// TIA Portal V20 export
// export: Created 2026-04-28T10:05:06.6637609Z, ExportSetting WithDefaults, DisplayName Totally Integrated Automation Portal, DisplayVersion V20, DisplayName TIA Portal Openness, DisplayVersion V20, DisplayName TIA Portal Version Control Interface, DisplayVersion V20, DisplayName SINAMICS Startdrive Advanced, DisplayVersion V20, DisplayName SINAMICS Startdrive G130, G150, S120, S150, SINAMICS MV, G220, S200, S210, DisplayVersion V20, DisplayName SINAMICS Startdrive G110M, G120, G120C, G120D, G120P, G115D, DisplayVersion V20, DisplayName STEP 7 Professional, DisplayVersion V20, DisplayName STEP 7 Safety, DisplayVersion V20, DisplayName WinCC Basic/Comfort/Advanced, DisplayVersion V20, DisplayName WinCC Unified, DisplayVersion V20
TYPE "REZEPT_VisuDaten"
TITLE = Rezeptdaten-Visualisierung
// Dieser Datentyp beinhaltet alle nötigen Daten für die Visualisierung.
// stored: IsFailsafeCompliant false
   STRUCT
      txt_rHotAirSoll : DInt;   // Set Value Hot air
      txt_rHotAirSt1 : DInt;   // Set Value Hot air level 1
      txt_rHotAirSt2 : DInt;   // Set Value Hot air level 2
      txt_rHotAirSt3 : DInt;   // Set Value Hot air level 3
      txt_rHotAirSt4 : DInt;   // Set Value Hot air level 4
      txt_rAlHoAi : DInt;   // Alarm Hot air
      txt_max_rDiPrFiBu : DInt;   // Differential pressure filter heating Input Limit
      txt_rDeliFan : DInt;   // Set Value Deli.Fan
      txt_rMinHotAirTempMainOff : DInt;   // Hot air temperature Min. for main fan off
      tTimeSt1 : Time;   // Timer Set Value Step 1
      tTimeSt2 : Time;   // Timer Set Value Step 2
      tTimeSt3 : Time;   // Timer Set Value Step 3
      txt_rPrToCtrl_Up : DInt := 0;   // Selection Negative pressure tower monitoring at defined intervals Up
      txt_rPrToCtrl_Down : DInt := 0;   // Selection Negative pressure tower monitoring at defined intervals Below
      txt_rPrToMa : DInt := 0;   // Pressure in tower Limit
      t_iKnValve_Gr1 : Time := T#0MS;   // Knock valves group 1 switch-on time
      t_iKnBreake_Gr1 : Time := T#0MS;   // Knock valves group 1 pause time
      t_iKnValve_Gr2 : Time := T#0MS;   // Knock valves group 2 switch-on time
      t_iKnBreake_Gr2 : Time := T#0MS;   // Knock valves group 2 pause time
      i_rExAiTe : DInt;   // Exhaust air Temperature Cleaning
      i_rHoAiTe : DInt;   // Hot air temperature Cleaning
      txt_rReGrHuMa : DInt := 0;   // Residual granulate humidity max.
      txt_rReGrHuSoll : DInt := 0;   // Residual granulate humidity Set Value
      txt_rGrTeCtrl_Up : DInt := 0;   // Selection Granulate Temperature monitoring at defined intervals Up
      txt_rGrTeCtrl_Down : DInt := 0;   // Selection Granulate Temperature monitoring at defined intervals Below
      txt_rGrTeMa : DInt := 0;   // Granule temperature limit
      t_iTwPeVaTopOp : Time := T#0MS;   // Double pendulum flap 1 open
      t_iTwPeVaBotOp : Time := T#0MS;   // Double pendulum flap 2 open
      txt_rWarn_1 : DInt := 0;   // Bin 1 Fill warning in %
      txt_rEmpBin_1 : DInt := 0;   // Bin 1 empty
      txt_rFullBin_1 : DInt := 0;   // Bin 1 Full
      txt_CoWaFlCo : DInt := 0;   // Min. flow rate
      t_iPolyCoOn_ON : Time;   // Polyconveyor ON
      t_iPolyCoOn_OFF : Time;   // Polyconveyor OFF
      rBinLeMonitorSet : Real;   // SetValue Level measurement
      txt_rDiDuFiBa : DInt := 0;   // Alarm Value Differential pressure filter dust return
      txt_rPrede : DInt := 0;   // Set value Dust conveying fan
      t_iKnValve_1 : Time := T#0MS;   // Knock Valve on, Cyklon
      t_iKnBreake_1 : Time := T#0MS;   // Knock Valve Breake, Cyklon
      txt_rCyclone : DInt := 0;   // Selection Cyclone 1 or 2
      txt_rReturn : DInt := 0;   // Return or Bin
      txt_rFlRaCy : DInt;   // Max. Value Cyclone flow monitoring dust return
      xKnVaAuto_Gr3_HMI : Bool;   // Start knock valves group Module 40 HMI
      txt_rExAiTe : DInt := 0;   // Set Value extract air temperature (control)
      txt_rAlExAi : DInt := 0;   // Alarm Exhaust air Valve to open
      txt_rExAiVa : DInt := 0;   // Exhaust air Valve to close
      txt_rExAiMa : DInt := 0;   // Exhaust air max. Burner off
      txt_rExAiSl : DInt := 0;   // Exhaust air Slip pump on
      txt_rExAi_min : DInt := 0;   // Exhaust air temperature below Min
      txt_rPrCyMa : DInt := 0;   // Pressure in cyclone Max.
      txt_rDiPrFiMa : DInt := 0;   // Differential pressure filter Max.
      txt_rMaxDuFiMo : DInt := 0;   // Dust filter Monitoring Max.
      txt_rDiPrSucFiMa : DInt := 0;   // Differential pressure Filter Max.
      txt_rMainFanFU : DInt := 0;   // Set Value Main fan
      t_iKnValve_1_50 : Time := T#0MS;   // Knocker valves filter On
      t_iKnBreake_1_50 : Time := T#0MS;   // Knocker valves filter pause
      t_iFiValve_On : Time := T#0MS;   // Filter cleaning valves With = 1 / Without = 0 Time ON
      t_iFiValveBrake : Time := T#0MS;   // Filter cleaning valves With = 1 / Without = 0 Time break
      txt_rMinProAir : DInt := 0;   // Min. Process Air available
      xKnVaAuto_Gr4_HMI : Bool;   // Start knock valves group Module 50 HMI
      xOptFiVa_Activ : Bool;   // Filter cleaning valves activation
      txt_rPrCyCtrl_Down : DInt := 0;   // Selection Negative pressure Cyclone monitoring at defined intervals Below
      txt_rPrCyCtrl_Up : DInt := 0;   // Selection Negative pressure Cyclone monitoring at defined intervals Up
      txt_rDiPrFiCtrl_Up : DInt := 0;   // Selection Differential pressure filter monitoring at defined intervals Up
      txt_rDiPrFiCtrl_Down : DInt := 0;   // Selection Differential pressure filter monitoring at defined intervals Below
      txt_rExAiTeCtrl_Up : DInt := 0;   // Selection Exhaust air temperature monitoring monitoring at defined intervals Up
      txt_rExAiTeCtrl_Down : DInt := 0;   // Selection Exhaust air temperature monitoring monitoring at defined intervals Below
      txt_PrFLRaCtrl_Up : DInt := 0;   // Slip quantity monitoring at defined intervals Up
      txt_PrFLRaCtrl_Down : DInt := 0;   // Slip quantity monitoring at defined intervals Below
      txt_rPrSlCtrl_Up : DInt := 0;   // Slip pressure monitoring at defined intervals Up
      txt_rPrSlCtrl_Down : DInt := 0;   // Slip pressure monitoring at defined intervals Below
      txt_rPrSlMa : DInt := 0;   // Slip pressure Max
      txt_rFlRaMa : DInt := 0;   // Mass flow Max.
      txt_iTankLevMax : DInt := 0;   // Tank Level Max.
      txt_iTankLevMin : DInt := 0;   // Tank Level Min.
      txt_rCoAiMi : DInt := 0;   // Air flow nozzle Max.
      txt_cSlPu_1_2 : DInt := 0;   // Selection Slip Pump 1 or 2
      txt_rSlPu : DInt := 0;   // Set value Slip pump
      txt_rSlPu2 : DInt := 0;   // Set value Slip pump 2
      iSpOelTemp_1 : DInt := 0;   // Switching point 1 oil temperature slip pump
      iSpOelTemp_2 : DInt := 0;   // Switching point 2 oil temperature slip pump
      txt_PrSlControll : DInt := 0;   // Slip pressure (control)
      txt_PrSlToleranze : DInt := 0;   // Slip pressure (tolerance)
      rDiffSl1Sl2_Set : DInt := 0;   // Difference value of slip pressure 1 and 2
      txt_rSlTeMa : DInt;   // Slip Temperature Max.
      txt_iPrSlTime : Time := T#0MS;   // Slip pressure Delay time
   END_STRUCT;
END_TYPE
